(* IEC 61131-3 sources: plc_generation_empirical_study/datasets/_archive/pre_native_plcverif_20260810/tasks/C01_E01_two_input_permissive/negative_control, 1 file *)

(* ---- NC1.st ---- *)
FUNCTION_BLOCK C01_E01_two_input_permissive
VAR_INPUT
    Enable : BOOL;
    GuardClosed : BOOL;
END_VAR
VAR_OUTPUT
    RunPermit : BOOL;
END_VAR

RunPermit := Enable OR GuardClosed;

END_FUNCTION_BLOCK
